PROGRAM LD_Example
VAR
END_VAR
VAR // added by the converter: edge detectors and wires of the graphical bodies
    _rt1 : R_TRIG;
END_VAR

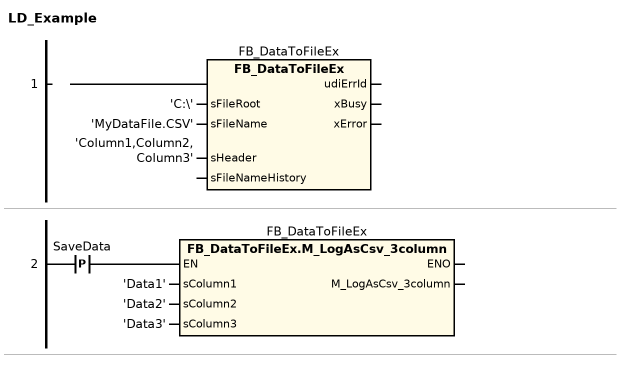
// NETWORK 1
FB_DataToFileEx(sFileRoot := 'C:\', sFileName := 'MyDataFile.CSV', sHeader := 'Column1,Column2,Column3');

// NETWORK 2
_rt1(CLK := SaveData);
IF _rt1.Q THEN
    FB_DataToFileEx.M_LogAsCsv_3column(sColumn1 := 'Data1', sColumn2 := 'Data2', sColumn3 := 'Data3');
END_IF

END_PROGRAM

(* stored: Version 1.1.0.1, ProductVersion 3.1.4020.6
   POU LD_Example: Id {ed28d828-0025-453a-b38b-73fba119846f}, SpecialFunc None *)
